Yaskawa INFORM job: R1_W53-A5(180,0)KM-OK_R2.JBI

/JOB
//NAME R1_W53-A5(180,0)KM-OK_R2
///FOLDERNAME KRIS-SCIANA
//POS
///NPOS 87,87,0,5,0,0
///TOOL 0
///POSTYPE PULSE
///PULSE
C00000=78189,-67986,-96830,-10467,37806,-7797
C00001=92440,-137165,-107216,-20191,-1154,-30432
C00002=111577,-35149,-80569,-22357,95949,-49570
C00003=108125,-69108,-70550,-21812,73585,-46669
C00004=108991,-69356,-70674,-22071,73765,-46380
C00005=108125,-69108,-70550,-21812,73585,-46669
C00006=108125,-69262,-73241,-21661,75055,-46942
C00007=117621,-69605,-71434,-24403,76492,-43697
C00008=117621,-69169,-67484,-24619,74475,-43270
C00009=117621,-69037,-66607,-24672,74044,-43177
C00010=117621,-69169,-67484,-24619,74475,-43270
C00011=115999,-31134,-49610,-23545,81846,-45382
C00012=115999,-31400,-47505,-23618,80529,-45120
C00013=115999,-31459,-46862,-23643,80137,-45042
C00014=115999,-31400,-47505,-23618,80529,-45120
C00015=106921,-27663,-53003,-20753,83100,-48803
C00016=107222,-27278,-49731,-20915,81470,-48417
C00017=107766,-27477,-49868,-21082,81586,-48247
C00018=107222,-27278,-49731,-20915,81470,-48417
C00019=104533,-24719,-53390,-19957,84187,-49799
C00020=110426,60287,26351,-21958,80569,-47129
C00021=110908,59737,28253,-22180,79343,-46729
C00022=111296,59567,28059,-22288,79474,-46610
C00023=110908,59737,28253,-22180,79343,-46729
C00024=110908,60137,25758,-22083,80961,-47030
C00025=115927,58509,23912,-23487,82578,-45556
C00026=115927,57802,29550,-23693,79052,-44852
C00027=115927,57770,30408,-23730,78553,-44752
C00028=115927,57802,29550,-23693,79052,-44852
C00029=115438,37086,-3507,-23221,87854,-46757
C00030=105503,-62969,-89657,-20228,86421,-49842
C00031=110518,-93811,-72284,-25294,103379,-67006
C00032=109543,-97011,-70118,-25208,100377,-66720
C00033=109125,-98154,-69170,-25203,99187,-66619
C00034=109125,-97062,-67033,-25140,98501,-66471
C00035=109125,-98154,-69170,-25203,99187,-66619
C00036=109271,-97171,-69065,-25206,99632,-66661
C00037=108845,-100765,-70348,-25219,98541,-66586
C00038=109271,-97171,-69065,-25206,99632,-66661
C00039=102810,-100484,-71733,-21889,96863,-67504
C00040=105287,-101169,-71975,-21344,97318,-66684
C00041=102810,-100484,-71733,-21889,96863,-67504
C00042=103151,-99431,-72768,-21891,98051,-67597
C00043=103951,-96443,-75155,-21958,101060,-67861
C00044=107257,-100648,-73272,-10850,107469,-69930
C00045=107258,-98768,-69563,-10763,106175,-69811
C00046=112732,-102414,-73458,-8827,107350,-67938
C00047=107259,-98817,-69673,-10765,106216,-69815
C00048=107581,-95618,-67198,-10659,106378,-69713
C00049=107132,-98744,-68135,-10755,105306,-69778
C00050=109929,-96120,-62444,-33323,94527,-78187
C00051=106572,-95477,-62214,-34043,93376,-79177
C00052=105781,-95731,-62292,-31308,97836,-75763
C00053=108056,-94926,-62112,-24163,105722,-68769
C00054=107208,-94572,-61089,-27775,101795,-84365
C00055=107266,-95021,-62493,-27833,102377,-84485
C00056=107266,-96693,-65652,-27971,103342,-84724
C00057=122843,-112109,-94588,-24450,117159,-81729
C00058=129835,-134677,-103725,-23924,94621,-78436
C00059=122031,-142599,-115737,-21891,54369,-80547
C00060=98554,-52920,-74241,8189,75358,-88961
C00061=99929,-44966,-62688,7728,72234,-88702
C00062=100515,-41335,-58144,8742,67143,-88703
C00063=99407,-48677,-66410,9194,68560,-88986
C00064=91136,-84016,-84009,13782,62520,-84975
C00065=92185,-81914,-79499,13487,60699,-84790
C00066=94678,-69213,-73775,11937,63247,-83539
C00067=92282,-85762,-85848,13207,62564,-84525
C00068=96355,-62297,-82866,4418,90457,-81939
C00069=96141,-62874,-78206,4448,87330,-82117
C00070=94818,-78572,-84878,4760,83458,-82696
C00071=94818,-78159,-88230,4747,85725,-82609
C00072=92917,-100987,-93906,5256,77635,-83573
C00073=92891,-101085,-92568,5277,76768,-83619
C00074=91442,-116772,-96989,5738,71551,-84363
C00075=89952,-133453,-104528,6223,67750,-85090
C00076=88868,-140609,-101302,6763,62208,-85804
C00077=87560,-150556,-102897,7361,58216,-86556
C00078=87221,-157626,-103100,7743,54770,-86930
C00079=90558,-160218,-104435,6930,53974,-85671
C00080=146191,-151469,-95869,-30859,62420,-61537
C00081=106395,-169325,-101560,-4487,45646,-78158
C00082=112535,-163276,-100430,-6672,52202,-75856
C00083=139479,-161729,-100194,-12010,55778,-65719
C00084=107096,-171190,-106994,-4543,48059,-77981
C00085=118025,-147103,-122296,-20754,32567,-81607
C00086=60212,-150278,-123121,-19822,31163,79382
BC00000=191480,536725,1075165
BC00001=211047,492979,1075167
BC00002=219137,444271,1075169
BC00003=219137,420955,1075169
BC00004=219137,420955,1075169
BC00005=219137,420955,1075169
BC00006=219137,420955,1075169
BC00007=219137,420955,1075169
BC00008=219137,420955,1075169
BC00009=219137,420955,1075169
BC00010=219137,420955,1075169
BC00011=219137,420955,1075169
BC00012=219137,420955,1075169
BC00013=219137,420955,1075169
BC00014=219137,420955,1075169
BC00015=219137,420955,1075169
BC00016=219137,420955,1075169
BC00017=219137,420955,1075169
BC00018=219137,420955,1075169
BC00019=219137,420955,1075169
BC00020=219137,459573,1075169
BC00021=219137,459573,1075169
BC00022=219137,459573,1075169
BC00023=219137,459573,1075169
BC00024=219137,459573,1075169
BC00025=219137,459573,1075169
BC00026=219137,459573,1075169
BC00027=219137,459573,1075169
BC00028=219137,459573,1075169
BC00029=219137,459573,1075169
BC00030=219137,444271,1075169
BC00031=237082,336217,1075175
BC00032=237082,336217,1075175
BC00033=237082,336217,1075175
BC00034=237082,336217,1075175
BC00035=237082,336217,1075175
BC00036=237082,336217,1075175
BC00037=237082,336217,1075175
BC00038=237082,336217,1075175
BC00039=237082,336217,1075175
BC00040=237082,336217,1075175
BC00041=237082,336217,1075175
BC00042=237082,336217,1075175
BC00043=237082,336217,1075175
BC00044=264111,319273,1075175
BC00045=262937,324659,1075175
BC00046=262467,326813,1075175
BC00047=262467,326813,1075175
BC00048=262467,326813,1075175
BC00049=262467,326813,1075175
BC00050=226039,338594,1075175
BC00051=226039,338594,1075175
BC00052=234841,330773,1075175
BC00053=257071,323674,1075171
BC00054=249909,329515,1075175
BC00055=249045,327149,1075175
BC00056=246884,321232,1075175
BC00057=246884,321232,1075175
BC00058=246884,321232,1075175
BC00059=246884,356761,1075175
BC00060=246884,356761,1075175
BC00061=246884,356761,1075175
BC00062=246884,356761,1075175
BC00063=246884,356761,1075175
BC00064=246884,356761,1075175
BC00065=246886,356761,1075173
BC00066=246886,356761,1075173
BC00067=246886,356761,1075173
BC00068=246886,356761,1075173
BC00069=246886,356761,1075171
BC00070=246886,356761,1075171
BC00071=246886,356761,1075171
BC00072=246886,356761,1075171
BC00073=246886,356761,1075171
BC00074=246886,356761,1075171
BC00075=246886,356761,1075171
BC00076=246886,356761,1075171
BC00077=246886,356761,1075171
BC00078=246886,356761,1075171
BC00079=246886,356761,1075171
BC00080=246886,356761,1075171
BC00081=246886,356761,1075171
BC00082=246886,356761,1075171
BC00083=246886,356761,1075171
BC00084=246886,356761,1075171
BC00085=246884,376000,1075175
BC00086=208302,536639,1074746
///POSTYPE BASE
///RECTAN
///RCONF 0,0,0,0,1,0,0,0,0,0,0,0,0,0,0,0,0,0,0,0,0,0,0,0
P00006=2.006,1.622,-0.565,0.0000,0.0000,0.0000
///RCONF 0,0,0,0,0,0,0,0,0,0,0,0,0,0,0,0,0,0,0,0,0,0,0,0
P00023=-2.957,-4.083,2.762,0.0000,0.0000,0.0000
P00025=3.643,0.007,-2.585,0.0000,0.0000,0.0000
P00026=2.644,0.055,-2.583,0.0000,0.0000,0.0000
P00027=2.278,0.099,-4.210,0.0000,0.0000,0.0000
//INST
///DATE 2024/06/10 13:13
///ATTR SC,RW
///GROUP1 RB1,BS1
NOP
'r2_W53-A5(180,0)
'Path S1074
MOVJ C00000 BC00000 VJ=20.00
SFTOF
MOVJ C00001 BC00001 VJ=10.00
MOVJ C00002 BC00002 VJ=10.00
MOVJ C00003 BC00003 VJ=10.00
REFP 3 C00004 BC00004
CALL JOB:SEARCH-R1
SET P025 P006
SFTON P025
MOVL C00005 BC00005 V=60.0
MOVL C00006 BC00006 V=100.0
MOVL C00007 BC00007 V=100.0
MOVL C00008 BC00008 V=100.0
REFP 3 C00009 BC00009
CALL JOB:SEARCH-R1
SET P025 P006
SFTON P025
MOVL C00010 BC00010 V=60.0
SFTOF
MOVL C00011 BC00011 V=100.0
MOVL C00012 BC00012 V=100.0
REFP 3 C00013 BC00013
CALL JOB:SEARCH-R1
SET P026 P006
SFTON P026
MOVL C00014 BC00014 V=60.0
MOVL C00015 BC00015 V=100.0
MOVL C00016 BC00016 V=100.0
REFP 3 C00017 BC00017
CALL JOB:SEARCH-R1
SET P026 P006
SFTON P026
MOVL C00018 BC00018 V=60.0
MOVL C00019 BC00019 V=100.0
MOVL C00020 BC00020 V=100.0
MOVL C00021 BC00021 V=100.0
REFP 3 C00022 BC00022
CALL JOB:SEARCH-R1
SET P027 P006
SFTON P027
MOVL C00023 BC00023 V=60.0
MOVL C00024 BC00024 V=100.0
MOVL C00025 BC00025 V=100.0
MOVL C00026 BC00026 V=100.0
REFP 3 C00027 BC00027
CALL JOB:SEARCH-R1
SET P027 P006
SFTON P027
MOVL C00028 BC00028 V=60.0
MOVJ C00029 BC00029 VJ=10.00
MOVJ C00030 BC00030 VJ=10.00
MOVJ C00031 BC00031 VJ=20.00
MOVL C00032 BC00032 V=100.0
MOVL C00033 BC00033 V=60.0
REFP 3 C00034 BC00034
CALL JOB:SEARCH-R1
SET P023 P006
SFTON P023
MOVL C00035 BC00035 V=60.0
MOVL C00036 BC00036 V=60.0
REFP 3 C00037 BC00037
CALL JOB:SEARCH-R1
SET P023 P006
SFTON P023
MOVL C00038 BC00038 V=60.0
MOVL C00039 BC00039 V=60.0
REFP 3 C00040 BC00040
CALL JOB:SEARCH-R1
SET P023 P006
SFTON P023
MOVL C00041 BC00041 V=60.0
MOVL C00042 BC00042 V=100.0
MOVL C00043 BC00043 V=100.0
'Path W1075
SFTOF
MOVJ C00044 BC00044 VJ=20.00
MOVL C00045 BC00045 V=100.0
SFTON P023
MOVL C00046 BC00046 V=100.0 PL=0
REFP 1 C00047 BC00047
REFP 2 C00048 BC00048
MACRO1 MJ#(0) ARGF9
ARCON
MOVL C00049 BC00049 V=10.0
MOVL C00050 BC00050 V=8.3
MOVL C00051 BC00051 V=8.3
MOVL C00052 BC00052 V=8.3
MOVL C00053 BC00053 V=8.3
MOVL C00054 BC00054 V=8.3
ARCOF
MOVL C00055 BC00055 V=100.0
MOVL C00056 BC00056 V=100.0
MOVJ C00057 BC00057 VJ=20.00
MOVJ C00058 BC00058 VJ=20.00
SFTOF
MOVJ C00059 BC00059 VJ=50.00
MOVJ C00060 BC00060 VJ=50.00
SFTON P027
MACRO1 MJ#(0) ARGF6
MOVJ C00061 BC00061 VJ=15.00
ARCON
MOVL C00062 BC00062 V=13.3
ARCOF
MOVJ C00063 BC00063 VJ=15.00
MOVJ C00064 BC00064 VJ=15.00
MOVJ C00065 BC00065 VJ=15.00
ARCON
MOVL C00066 BC00066 V=13.3
ARCOF
MOVJ C00067 BC00067 VJ=15.00
SFTOF
MOVJ C00068 BC00068 VJ=15.00
SFTON P026
MOVJ C00069 BC00069 VJ=15.00
ARCON
MOVL C00070 BC00070 V=13.3
ARCOF
MOVJ C00071 BC00071 VJ=15.00
MOVJ C00072 BC00072 VJ=15.00
MOVJ C00073 BC00073 VJ=15.00
ARCON
MOVL C00074 BC00074 V=13.3
ARCOF
MOVJ C00075 BC00075 VJ=15.00
SFTOF
SFTON P025
MOVJ C00076 BC00076 VJ=15.00
ARCON
MOVL C00077 BC00077 V=13.3
MOVL C00078 BC00078 V=13.3
ARCOF
MOVJ C00079 BC00079 VJ=15.00
MOVL C00080 BC00080 V=83.3
ARCON
MOVL C00081 BC00081 V=13.3
MOVL C00082 BC00082 V=13.3
MACRO1 MJ#(0) ARGF12
ARCON
WVON WEV#(50)
MOVL C00083 BC00083 V=13.3
ARCOF
WVOF
SFTOF
MOVJ C00084 BC00084 VJ=15.00
MOVJ C00085 BC00085 VJ=20.00
MOVJ C00086 BC00086 VJ=100.00
SFTOF
END
